TYPE PWMControlChannel :
STRUCT
	{attribute addProperty Name "Control"}
	Control AT %Q* : stPWMcontrol;
	{attribute addProperty Name "PWM Output"}
	PWMOutput AT %Q* : INT;
END_STRUCT
END_TYPE

(* stored: Version 1.1.0.1, ProductVersion 3.1.4024.9
   DUT PWMControlChannel: Id {e2039fc0-c2b0-0a91-091b-0f12f7b7b5e4} *)
